// Mitsubishi GX Works2 project: Control Time Counting p102   PLC: FX3S
// Control Time Counting p102

PROGRAM MAIN
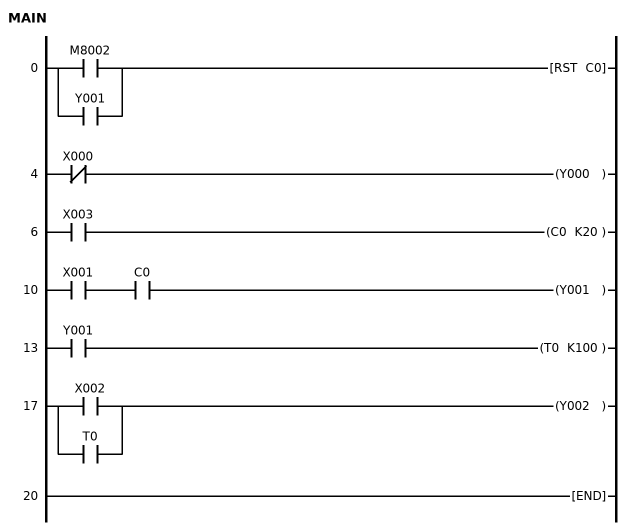
0     LD      M8002
      OR      Y001
      RST     C0
4     LDI     X000
      OUT     Y000
6     LD      X003
      OUT     C0 K20
10    LD      X001
      AND     C0
      OUT     Y001
13    LD      Y001
      OUT     T0 K100
17    LD      X002
      OR      T0
      OUT     Y002
20    END
END_PROGRAM
